// TIA Portal V17 export
// export: Created 2023-07-20T19:47:57.2444624Z, ExportSetting WithDefaults, DisplayName Totally Integrated Automation Portal, DisplayVersion V17 Update 4, DisplayName TIA Portal Openness, DisplayVersion V17 Update 4, DisplayName TIA Portal Teamcenter Gateway, DisplayVersion V17 Update 4, DisplayName TIA Portal Version Control Interface, DisplayVersion V17, DisplayName TIA Portal Test Suite Advanced, DisplayVersion V17, DisplayName SINAMICS Startdrive Advanced, DisplayVersion V17, DisplayName SINAMICS Startdrive G130, G150, S120, S150, SINAMICS MV, S210, DisplayVersion V17, DisplayName SINAMICS Startdrive G110M, G120, G120C, G120D, G120P, G115D, DisplayVersion V17, DisplayName STEP 7 Professional, DisplayVersion V17 Update 4, DisplayName SIMATIC Energy Suite, DisplayVersion V17, DisplayName STEP 7 Safety, DisplayVersion V17, DisplayName WinCC Advanced / Unified PC, DisplayVersion V17 Update 4, DisplayName SIMATIC Visualization Architect, DisplayVersion V17
ORGANIZATION_BLOCK "Startup"   // OB100, LAD, Startup
TITLE = "Complete Restart"
{ S7_Optimized_Access := 'TRUE' }
VERSION : 0.1
// stored: AutoNumber true, IsIECCheckEnabled false, SetENOAutomatically false
   VAR_INPUT
      LostRetentive : Bool;   // True if retentive data are lost
      LostRTC : Bool;   // True if date and time are lost
   END_VAR
   VAR_TEMP
      Flash : Bool;
   END_VAR
BEGIN

REGION Network 1: Stepper initial values
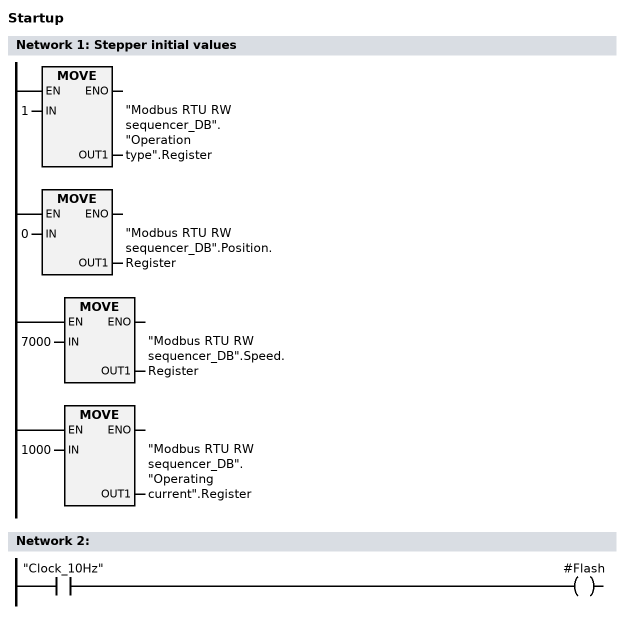
   RUNG wire#powerrail
      Move(in := 1, out1 => "Modbus RTU RW sequencer_DB"."Operation type".Register)
   END_RUNG
   RUNG wire#powerrail
      Move(in := 0, out1 => "Modbus RTU RW sequencer_DB".Position.Register)
   END_RUNG
   RUNG wire#powerrail
      Move(in := 7000, out1 => "Modbus RTU RW sequencer_DB".Speed.Register)
   END_RUNG
   RUNG wire#powerrail
      Move(in := 1000, out1 => "Modbus RTU RW sequencer_DB"."Operating current".Register)
   END_RUNG
   // the same network as SCL:
   "Modbus RTU RW sequencer_DB"."Operation type".Register := 1;
   "Modbus RTU RW sequencer_DB".Position.Register := 0;
   "Modbus RTU RW sequencer_DB".Speed.Register := 7000;
   "Modbus RTU RW sequencer_DB"."Operating current".Register := 1000;
END_REGION

REGION Network 2
   RUNG wire#powerrail
      Contact( "Clock_10Hz" )
      Coil( #Flash )
   END_RUNG
   // the same network as SCL:
   #Flash := "Clock_10Hz";
END_REGION
END_ORGANIZATION_BLOCK
